{attribute addProperty BoxType "EL6201-0000-0017"}
{attribute addProperty Id "Slave_7A_DO0BIT10.12549Slave_7A_DO1BIT10.12550Slave_7A_DO2BIT10.12551Slave_7A_DO3BIT10.12552Slave_7B_DO0BIT10.12553Slave_7B_DO1BIT10.12554Slave_7B_DO2BIT10.12555Slave_7B_DO3BIT10.12556"}
{attribute addProperty CRC "177600794"}
{attribute addProperty SizeInBites "8"}
{attribute addProperty SizeInBytes "1"}
TYPE Slave_7_Outputs_0A95F91A :
STRUCT
	{attribute addProperty Name "Slave_7A_DO0"}
	Slave_7A_DO0 : BIT;
	{attribute addProperty Name "Slave_7A_DO1"}
	Slave_7A_DO1 : BIT;
	{attribute addProperty Name "Slave_7A_DO2"}
	Slave_7A_DO2 : BIT;
	{attribute addProperty Name "Slave_7A_DO3"}
	Slave_7A_DO3 : BIT;
	{attribute addProperty Name "Slave_7B_DO0"}
	Slave_7B_DO0 : BIT;
	{attribute addProperty Name "Slave_7B_DO1"}
	Slave_7B_DO1 : BIT;
	{attribute addProperty Name "Slave_7B_DO2"}
	Slave_7B_DO2 : BIT;
	{attribute addProperty Name "Slave_7B_DO3"}
	Slave_7B_DO3 : BIT;
END_STRUCT
END_TYPE

(* stored: Version 1.2.0.0, ProductVersion 3.1.4024.9
   DUT Slave_7_Outputs_0A95F91A: Id {114f2eed-5618-4fba-9695-9419969180bd} *)
